(*

.. <legal notes>

legal notes
=================
| SPDX-FileCopyrightText: © 2025 Oleksandr Tiutyk <trofimich@gmail.com>
| SPDX-License-Identifier: LGPL-3.0-only
| For details check: LGPL-3.0-only_

.. _LGPL-3.0-only: https://www.gnu.org/licenses/lgpl-3.0.en.html

.. </legal notes>

*)

FUNCTION_BLOCK TrafficLight EXTENDS TOF_Automation.OutputDevice<3>
VAR_OUTPUT
	RedLight : TOF_Devices_IO.DigitalOutput(THIS^, CONTACT_TYPE.NORMALY_OPEN);
	YellowLight : TOF_Devices_IO.DigitalOutput(THIS^, CONTACT_TYPE.NORMALY_OPEN);
	GreenLight : TOF_Devices_IO.DigitalOutput(THIS^, CONTACT_TYPE.NORMALY_OPEN);
END_VAR
VAR
	_ClassName : STRING := __POUNAME();
	
	_SubDevices : ARRAY [0..2] OF TOF_Automation.IDevice := [RedLight, YellowLight, GreenLight];
END_VAR

{attribute 'monitoring' := 'call'}
PROPERTY ClassName : STRING
GET
ClassName := _ClassName;
END_GET
END_PROPERTY

METHOD PROTECTED OnUpdateOutputsFromState
VAR_IN_OUT CONSTANT
	executionContext : TOF_Automation.AUTOMATION_EXECUTION_CONTEXT;
END_VAR
// No additional logic here
END_METHOD

METHOD SetLight
VAR_INPUT
	color : TRAFFIC_LIGHT_COLOR;
END_VAR
RedLight.Value := color = TRAFFIC_LIGHT_COLOR.RED;
YellowLight.Value := color = TRAFFIC_LIGHT_COLOR.YELLOW;
GreenLight.Value := color = TRAFFIC_LIGHT_COLOR.GREEN;
END_METHOD

{attribute 'monitoring' := 'call'}
PROPERTY Size : ULINT
GET
Size := XSIZEOF(THIS^);
END_GET
END_PROPERTY

PROPERTY SubDevices : REFERENCE TO ARRAY [0..(_SubDeviceCount_ - 1)] OF TOF_Automation.IDevice
GET
SubDevices REF= _SubDevices;
END_GET
END_PROPERTY

END_FUNCTION_BLOCK

(* stored: Version 1.1.0.1
   POU TrafficLight: Id {4a48deea-1b31-43e8-87e2-aa154a1466e2}, SpecialFunc None
   Property ClassName: Id {57d4725e-1474-4661-8746-ce344608dbc4}
   Get Get: Id {bf033ab4-a042-404c-85bc-755e1b6f3d73}
   Method OnUpdateOutputsFromState: Id {e35a0913-4b43-401c-adae-5085684557d7}
   Method SetLight: Id {66ac2472-cd7a-4221-b0c7-b8380631be67}
   Property Size: Id {0854c0b6-08bb-4062-b879-abc7c2048c2f}
   Get Get: Id {be673c01-8bac-444a-bd16-fa3be540c5df}
   Property SubDevices: Id {24d9159e-d58e-4242-9c68-13fddc2a3388}
   Get Get: Id {a8e5d14a-9275-4393-b35e-1978fe96fc18} *)
